FUNCTION_BLOCK PhaseObjTestBasic (* Basic Function Block Type *)
  (* Standard: 61499-2 *)
  (* Version 0.0, 6/5/2026, Schneider Electric, Template *)
  PACKAGE SE.Nereda;
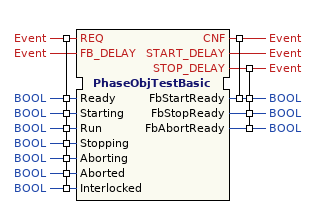
  EVENT_INPUT
    REQ WITH Starting, Stopping, Aborting, Ready, Run, Aborted, Interlocked; (* Normal Execution Request *)
    FB_DELAY;
  END_EVENT
  EVENT_OUTPUT
    CNF WITH FbStartReady; (* Execution Confirmation *)
    START_DELAY;
    STOP_DELAY WITH FbStartReady, FbStopReady, FbAbortReady;
  END_EVENT
  VAR_INPUT
    Ready : BOOL;
    Starting : BOOL;
    Run : BOOL;
    Stopping : BOOL;
    Aborting : BOOL;
    Aborted : BOOL;
    Interlocked : BOOL;
  END_VAR
  VAR_OUTPUT
    FbStartReady : BOOL;
    FbStopReady : BOOL;
    FbAbortReady : BOOL;
  END_VAR
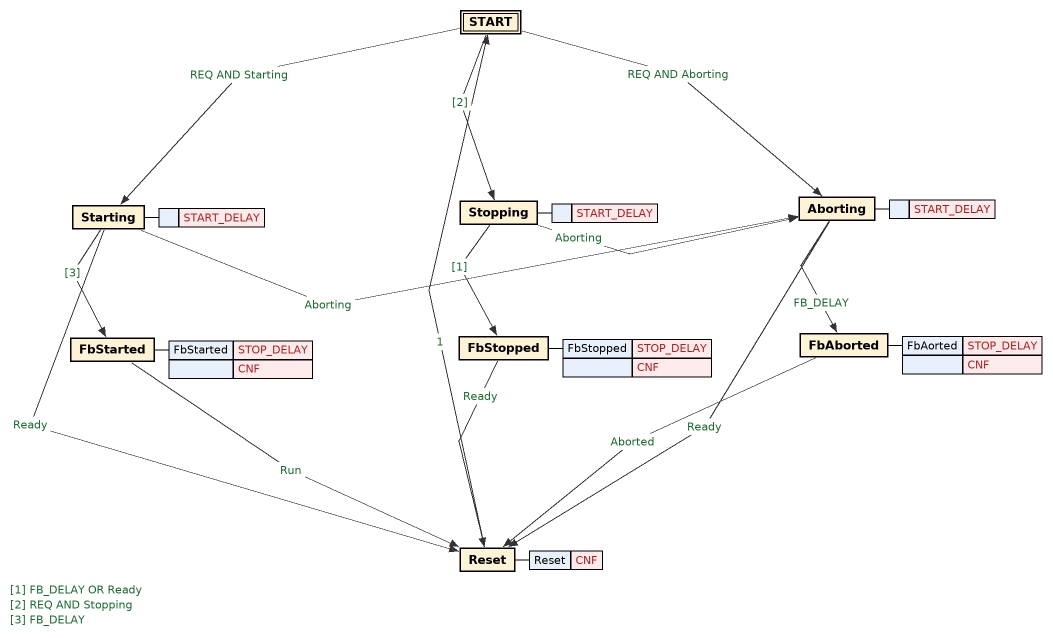
  EC_STATES
    START; (* Initial State *)
    Starting : -> START_DELAY;
    FbStarted : FbStarted -> STOP_DELAY, -> CNF;
    Stopping : -> START_DELAY;
    FbStopped : FbStopped -> STOP_DELAY, -> CNF;
    Aborting : -> START_DELAY;
    FbAborted : FbAorted -> STOP_DELAY, -> CNF;
    Reset : Reset -> CNF;
  END_STATES
  EC_TRANSITIONS
    START TO Aborting := REQ AND Aborting;
    START TO Stopping := REQ AND Stopping;
    START TO Starting := REQ AND Starting;
    Aborting TO FbAborted := FB_DELAY;
    Starting TO FbStarted := FB_DELAY;
    Stopping TO FbStopped := FB_DELAY OR Ready;
    FbStarted TO Reset := Run;
    FbStopped TO Reset := Ready;
    FbAborted TO Reset := Aborted;
    Reset TO START := 1;
    Starting TO Aborting := Aborting;
    Stopping TO Aborting := Aborting;
    Starting TO Reset := Ready;
    Aborting TO Reset := Ready;
  END_TRANSITIONS
  ALGORITHM FbStarted IN ST:
;
FbStartReady := TRUE;
FbStopReady := FALSE;
FbAbortReady := FALSE;
  END_ALGORITHM
  ALGORITHM FbStopped IN ST:
;
FbStartReady := FALSE;
FbStopReady := TRUE;
FbAbortReady := FALSE;
  END_ALGORITHM
  ALGORITHM FbAorted IN ST:
;
FbStartReady := FALSE;
FbStopReady := FALSE;
FbAbortReady := TRUE;
  END_ALGORITHM
  ALGORITHM Reset IN ST:
;
FbStartReady := FALSE;
FbStopReady := FALSE;
FbAbortReady := FALSE;
  END_ALGORITHM
END_FUNCTION_BLOCK
